// TwinCAT 3 PLC project Punzonatrice01
// ProgramVersion: 3.1.4024.0
// libraries:
//   Tc2_Standard, * (Beckhoff Automation GmbH)
//   Tc2_System, * (Beckhoff Automation GmbH)
//   Tc3_Module, * (Beckhoff Automation GmbH)
//   Util, * (System)
// project tree:
//   DUTs/ tStatiMSF.TcTLEO
//   GVLs/ GVL_IO.TcGVL
//   / PlcTask.TcTTO
//   POUs/ MAIN.TcPOU
//   POUs/MSF/FB/ FB_Blink.TcPOU, FB_MSF.TcPOU
// real-time tasks:
//   TASK PlcTask: cycle T#10ms, priority 20, ADS port 350
// motion (NC):
//   TASK NC-Task 1 SAF: cycle T#2ms, priority 4, ADS port 501
//   TASK NC-Task 1 SVB: cycle T#10ms, priority 8, ADS port 511
//   AXIS Asse 1 (id 1)
//     OtherSettings: AllowMotionCmdToSlave=true
//     encoder EncType=4
//       EncPara: MaxCount=#x0000ffff
//         Inc: RefSoftSyncMask=#x0000ffff
//     drive DrvType=24
//       Analog: TorqueSetpointScale=10, ScaleFactorActTorque=0.1
//       TimeComp: TaskDelayCycles=1
//     controller CtrType=1
//       CtrPara: PriorControlFactor=1
//         Observer: BandWidth=20
// I/O:
//   DEVICE Dispositivo 1 (EtherCAT), AmsNetId 192.168.17.154.2.1
//     Terminale 1 (EK1200) [EK1200-5000 EtherCAT Power supply (2A E-Bus)]
//       Terminale 2 (EL1809) [EL1809 16Ch. Dig. Input 24V, 3ms]
//       Terminale 3 (EL2809) [EL2809 16Ch. Dig. Output 24V, 0.5A]
//       Terminale 4 (EL3201) [EL3201 1Ch. Ana. Input PT100 (RTD)]
//       Terminale 5 (EL3311) [EL3311 1Ch. Ana. Input Thermocouple (TC)]
//       Terminale 6 (EL3004) [EL3004 4Ch. Ana. Input +/-10V]
//       Terminale 7 (EL1918) [EL1918, 8Ch. Safety Input 24V, TwinSAFE]
//         modules: Module 1 (FSOE), Module 2 (FSLOGIC)
//       Terminale 8 (EL2904) [EL2904, 4 Ch. Safety Output 24V, 0.5A, TwinSAFE]
//         modules: Module 1 (FSOES), Module 2 (DO)
//       Terminale 9 (EL9011) [EL9011 End Terminal]
//   DEVICE Dispositivo 4 (EtherCAT), AmsNetId 192.168.17.154.5.1
//     Terminale 10 (EK1100) [EK1100 EtherCAT Coupler (2A E-Bus)]
//       Terminale 11 (EL1809) [EL1809 16Ch. Dig. Input 24V, 3ms]
//       Terminale 12 (EL2809) [EL2809 16Ch. Dig. Output 24V, 0.5A]
//       Terminale 13 (EL1809) [EL1809 16Ch. Dig. Input 24V, 3ms]
//       Terminale 14 (EL2809-0015) [EL2809-0015 16Ch. Dig. Output 24V DC, 0.35A, not short-circuit proof]
//       Terminale 15 (EL7031) [EL7031 1Ch. Stepper motor output stage (24V, 1.5A)]
//       Terminale 7 (EL9011) [EL9011 End Terminal]
// variable links:
//   NC-Task 1 SAF/Axes/Asse 1 <-> Device 4 (EtherCAT)/Term 10 (EK1100)/Term 15 (EL7031)
//     Drive/Inputs/In/nState1 @bit 3 <-> STM Status/Status/Error
//     Drive/Inputs/In/nState1 @bit 5 <-> STM Status/Status/Moving negative
//     Drive/Inputs/In/nState1 @bit 4 <-> STM Status/Status/Moving positive
//     Drive/Inputs/In/nState1 @bit 1 <-> STM Status/Status/Ready
//     Drive/Inputs/In/nState1 <-> STM Status/Status/Ready to enable
//     Drive/Inputs/In/nState1 @bit 6 <-> STM Status/Status/Torque reduced
//     Drive/Inputs/In/nState1 @bit 2 <-> STM Status/Status/Warning
//     Drive/Inputs/In/nState2 @bit 3 <-> STM Status/Status/Digital input 1
//     Drive/Inputs/In/nState2 @bit 4 <-> STM Status/Status/Digital input 2
//     Drive/Inputs/In/nState2 @bit 5 <-> STM Status/Status/Sync error
//     Drive/Inputs/In/nState2 @bit 7 <-> STM Status/Status/TxPDO Toggle
//     Drive/Inputs/In/nState4 @bit 1 <-> WcState/InputToggle
//     Drive/Inputs/In/nState4 <-> WcState/WcState
//     Drive/Outputs/Out/nCtrl1 <-> STM Control/Control/Enable
//     Drive/Outputs/Out/nCtrl1 @bit 2 <-> STM Control/Control/Reduce torque
//     Drive/Outputs/Out/nCtrl1 @bit 1 <-> STM Control/Control/Reset
//     Drive/Outputs/Out/nDataOut2[0] <-> STM Velocity/Velocity
//     Enc/Inputs/In/nDataIn1[0] <-> ENC Status compact/Counter value
//     Enc/Inputs/In/nDataIn2[0] <-> ENC Status compact/Latch value
//     Enc/Inputs/In/nState1 @bit 4 <-> ENC Status compact/Status/Counter overflow
//     Enc/Inputs/In/nState1 @bit 3 <-> ENC Status compact/Status/Counter underflow
//     Enc/Inputs/In/nState1 @bit 1 <-> ENC Status compact/Status/Latch extern valid
//     Enc/Inputs/In/nState1 @bit 2 <-> ENC Status compact/Status/Set counter done
//     Enc/Inputs/In/nState2 @bit 4 <-> ENC Status compact/Status/Status of extern latch
//     Enc/Inputs/In/nState2 @bit 5 <-> ENC Status compact/Status/Sync error
//     Enc/Inputs/In/nState2 @bit 7 <-> ENC Status compact/Status/TxPDO Toggle
//     Enc/Inputs/In/nState4 @bit 1 <-> WcState/InputToggle
//     Enc/Inputs/In/nState4 <-> WcState/WcState
//     Enc/Outputs/Out/nCtrl1 @bit 3 <-> ENC Control compact/Control/Enable latch extern on negative edge
//     Enc/Outputs/Out/nCtrl1 @bit 1 <-> ENC Control compact/Control/Enable latch extern on positive edge
//     Enc/Outputs/Out/nCtrl1 @bit 2 <-> ENC Control compact/Control/Set counter
//     Enc/Outputs/Out/nDataOut1[0] <-> ENC Control compact/Set counter value
//   Punzonatrice01/Punzonatrice01 Instance <-> Device 1 (EtherCAT)/Term 1 (EK1200)/Term 2 (EL1809)
//     PlcTask Inputs/GVL_IO.Ack <-> Channel 7/Input
//     PlcTask Inputs/GVL_IO.Emg <-> Channel 8/Input
//     PlcTask Inputs/GVL_IO.I{1..4} <-> Channel {1..4}/Input  (4 links)
//     PlcTask Inputs/GVL_IO.Start <-> Channel 5/Input
//     PlcTask Inputs/GVL_IO.Stop <-> Channel 6/Input
//   Punzonatrice01/Punzonatrice01 Instance <-> Device 1 (EtherCAT)/Term 1 (EK1200)/Term 3 (EL2809)
//     PlcTask Outputs/GVL_IO.L_ACK <-> Channel 7/Output
//     PlcTask Outputs/GVL_IO.L_START <-> Channel 5/Output
//     PlcTask Outputs/GVL_IO.L_STOP <-> Channel 6/Output
//     PlcTask Outputs/GVL_IO.Q{1..4} <-> Channel {1..4}/Output  (4 links)

CONFIGURATION Punzonatrice01
    RESOURCE PLC ON TwinCAT3
        TASK PlcTask(INTERVAL := T#10ms, PRIORITY := 20);
        PROGRAM MAIN WITH PlcTask : MAIN;
    END_RESOURCE
END_CONFIGURATION

// ---- DUTs/tStatiMSF.TcTLEO
{attribute 'qualified_only'}
{attribute 'strict'}
TYPE tStatiMSF :
(
	S0_Spento := 0,
	S1_RipristinoMandrino,
	S2_AttesaPezzo,
	S3_PausaIngresso,
	S4_Caricamento,
	S5_DiscesaMandrino,
	S6_SalitaMandrino,
	S7_Scarico,
	S8_PausaScarico,
	SE_Emergenza,
	SA1_RipristinoMAndrino,
	SA2_UscitaPezzo
);
END_TYPE

// ---- GVLs/GVL_IO.TcGVL
{attribute 'qualified_only'}
VAR_GLOBAL
	// sensori bordo macchina
    I1    AT %I*    :    BOOL;
    I2    AT %I*    :    BOOL;
    I3    AT %I*    :    BOOL;
    I4    AT %I*    :    BOOL;
    // pulsanti di comando
    Start    AT %I*    :    BOOL;
    Stop    AT %I*    :    BOOL;
    Ack        AT %I*    :    BOOL;
    Emg        AT %I*    :    BOOL;
 
    // attuatori
    Q1    AT %Q*    :    BOOL;
    Q2    AT %Q*    :    BOOL;
    Q3    AT %Q*    :    BOOL;
    Q4    AT %Q*    :    BOOL;
    // indicatori pannello operatore
    L_START    AT %Q*    :    BOOL;
    L_STOP    AT %Q*    :    BOOL;
    L_ACK    AT %Q*    :    BOOL;    
END_VAR

// ---- POUs/MAIN.TcPOU
PROGRAM MAIN
VAR
	nastro1	: FB_MSF();
	
END_VAR

nastro1(
	I1:= GVL_IO.I1, 
	I2:= GVL_IO.I2, 
	I3:= GVL_IO.I3, 
	I4:= GVL_IO.I4, 
	Start:= GVL_IO.Start, 
	Stop:= GVL_IO.Stop, 
	Ack:= GVL_IO.Ack, 
	Emg:= GVL_IO.Emg, 
	Q1=> GVL_IO.Q1, 
	Q2=> GVL_IO.Q2, 
	Q3=> GVL_IO.Q3, 
	Q4=> GVL_IO.Q4, 
	L_START=> GVL_IO.L_START, 
	L_STOP=> GVL_IO.L_STOP, 
	L_ACK=> GVL_IO.L_ACK);

END_PROGRAM

// ---- POUs/MSF/FB/FB_MSF.TcPOU
FUNCTION_BLOCK FB_MSF
VAR_INPUT
	// sensori bordo macchina
	I1		:	BOOL;
	I2		: 	BOOL;
	I3		:	BOOL;
	I4		: 	BOOL;
	
	// pulsanti di comando
	Start	: 	BOOL;
	Stop	:	BOOL;
	Ack		: 	BOOL;
	Emg		: 	BOOL;
	
END_VAR
VAR_OUTPUT
	// attuatori
	Q1		:	BOOL;
	Q2		:	BOOL;
	Q3		:	BOOL;
	Q4		:	BOOL;

	// indicatori pannello indicatore
	L_START	: 	BOOL;
	L_STOP	: 	BOOL;
	L_ACK	: 	BOOL;
END_VAR
VAR
	// abilitazione := Stop AND Emg;
	enable 	:	BOOL;
	
	// variabile di stato
	stato	:	tStatiMSF	:=	tStatiMSF.S0_Spento;
	
	// timer per gli stati
	T34		: 	TON();
	T82		:	TON();
	TE		:	TON();
	TA		:	TON();
	
	// lampeggiatore
	osc		: 	FB_Blink();
	fbBlink :   BLINK;
	// richiesta di arresto a fine ciclo
	mArresto	:	BOOL;

	// pezzo carico
	mPezzoCarico	:	BOOL;
	// transizione S0->S1
	tr_S0_S1	: 	BOOL;
	// transizione S0->S1
	tr_S0_S2	: 	BOOL;
	// transizione S1->S0
	tr_S1_S0	:	BOOL;
	// transizione S1->S2
	tr_S1_S2	: 	BOOL;
	//transizione da S2->S3
	tr_S2_S0	:	BOOL;
	// transizione S2->S3
	tr_S2_S3	: 	BOOL;
	// transizione S3->S4
	tr_S3_S4	: 	BOOL;
	// transizione S4->S5
	tr_S4_S5	: 	BOOL;
	// transizione S4->S5
	tr_S4_SE	: 	BOOL;
	// transizione S5->S6
	tr_S5_S6	: 	BOOL;
	// transizione S6->S7
	tr_S6_S7	: 	BOOL;
	// transizione S7->S8
	tr_S7_S8	: 	BOOL;
	// transizione S7->SE
	tr_S7_SE	: 	BOOL;
	// transizione S8->S0
	tr_S8_S0	: 	BOOL;
	// transizione S8->S2
	tr_S8_S2	: 	BOOL;
	// transizione SE->SA
	tr_SE_SA1	: 	BOOL;
	// transizione SA1->SA2
	tr_SA1_SA2	: 	BOOL;
	// transizione SA2->S0
	tr_SA2_S0	: 	BOOL;
END_VAR

// 1. aggiornamento delle condizioni di abilitazione (stop, allatmi, ecc)
	enable	:=	Stop AND Emg;
	
// 2. aggiornamento di timers, contatori, triggers sui fronti
	T34( IN := (stato = tStatiMSF.S3_PausaIngresso), PT := T#2S );
	T82( IN := (stato = tStatiMSF.S8_PausaScarico), PT := T#3S );
	TE( IN := (stato = tStatiMSF.S4_Caricamento), PT := T#5S );
	TE( IN := (stato = tStatiMSF.S7_Scarico), PT := T#5S );
	TE( IN := (stato = tStatiMSF.SA2_UscitaPezzo), PT := T#5S );
	TA( IN := (stato = tStatiMSF.SA1_RipristinoMandrino), PT := T#2S );
	osc(enable := TRUE, t_high := T#1S, t_low := T#500MS);
// 3. valutazione della condizione di arresto nominale
	IF( Stop = FALSE AND Emg = TRUE ) THEN 
		mArresto := TRUE;
	END_IF
	
// 4. valutazione della condizione di arresto di emergenza
	IF( Emg = FALSE AND (stato <> tStatiMSF.S0_Spento)) THEN
		stato := tStatiMSF.SE_Emergenza;
	END_IF
	
	
// 5. aggiornamento delle condizioni di transito di stato
	tr_S0_S1 :=	NOT(I3) AND Start AND enable;
	// transizione S0->S2
	tr_S0_S2 := I3 AND Start AND enable; 
	// transizione S1->S0
	tr_S1_S0 := mArresto AND Emg;	
	// transizione S1->S2
	tr_S1_S2 := I3 AND Emg;
	//transizione da S2->S3
	tr_S2_S0 := mArresto AND Emg;
	// transizione S2->S3
	tr_S2_S3 := NOT(I1) AND Emg;
	// transizione S3->S4
	tr_S3_S4 := T34.Q AND NOT(I1) AND Emg;
	// transizione S4->S5
	tr_S4_S5 := NOT(I2) AND Emg; 
	// transizione S4->S5
	tr_S4_SE := TE.Q AND Emg;	
	// transizione S5->S6
	tr_S5_S6 := I4 AND Emg; 
	// transizione S6->S7
	tr_S6_S7 := I3 AND Emg;
	// transizione S4->S5
	tr_S7_SE := TE.Q AND Emg;
	// transizione S7->S8
	tr_S7_S8 := NOT(I1) AND Emg;
	// transizione S8->S0
	tr_S8_S0 := mArresto AND Emg ;
	// transizione S8->S2
	tr_S8_S2 := T82.Q AND NOT(mArresto) AND I1 AND enable;
	// transizione SE->SA
	tr_SE_SA1 := EMG AND Ack;
	// transizione SE->SA
	tr_SA1_SA2 := TA.Q;
	// transizione SA->S0
	tr_SA2_S0 := (mPezzoCarico AND NOT(I1) AND I3) OR (NOT(mPezzoCarico) AND I3)OR(TE.Q);

// 6. switch-case della MSF
	CASE stato OF
	tStatiMSF.S0_Spento:
	

    // comando uscite
	L_START := FALSE;
	L_STOP := TRUE;
	L_ACK := FALSE;
	Q1 := FALSE;
	Q2 := FALSE;
	Q3 := FALSE;
	Q4 := FALSE;
	// reset memoria
	mArresto := FALSE;
	mPezzoCarico := FALSE;
	IF tr_S0_S1 THEN
		stato := tStatiMSF.S1_RipristinoMandrino;
	ELSIF tr_S0_S2 THEN
		stato := tStatiMSF.S2_AttesaPezzo;
	END_IF
	
	tStatiMSF.S1_RipristinoMandrino:
	// comando uscite
	L_START := TRUE;
	L_STOP := FALSE;
	L_ACK := osc.q;// lamepggio
	Q1 := FALSE;
	Q2 := FALSE;
	Q3 := NOT(I3);
	Q4 := FALSE;
	// set memoria
	mPezzoCarico := FALSE;
	IF tr_S1_S2 THEN
		stato := tStatiMSF.S2_AttesaPezzo;
	ELSIF tr_S1_S0 THEN
		stato := tStatiMSF.S0_Spento;
	END_IF
	
	tStatiMSF.S2_AttesaPezzo:
	// comando uscite
	L_START := TRUE;
	L_STOP := FALSE;
	L_ACK := FALSE;
	Q1 := FALSE;
	Q2 := FALSE;
	Q3 := FALSE;
	Q4 := FALSE;
	// set memoria
	mPezzoCarico := FALSE;
	IF tr_S2_S3 THEN
		stato := tStatiMSF.S3_PausaIngresso;
	ELSIF tr_S2_S0 THEN
		stato := tStatiMSF.S0_Spento;
	END_IF
	
	tStatiMSF.S3_PausaIngresso:
	// comando uscite
	L_START := TRUE;
	L_STOP := FALSE;
	L_ACK := FALSE;
	Q1 := FALSE;
	Q2 := FALSE;
	Q3 := FALSE;
	Q4 := FALSE;
	// set memoria
	mPezzoCarico := TRUE;
	IF tr_S3_S4 THEN
		stato := tStatiMSF.S4_Caricamento;
	END_IF
	
	tStatiMSF.S4_Caricamento:
	// comando uscite
	L_START := TRUE;
	L_STOP := FALSE;
	L_ACK := FALSE;
	Q1 := TRUE;
	Q2 := FALSE;
	Q3 := FALSE;
	Q4 := FALSE;
	// set memoria
	mPezzoCarico := TRUE;
	IF tr_S4_S5 THEN
		stato := tStatiMSF.S5_DiscesaMandrino;
	ELSIF tr_S4_SE THEN
		stato := tStatiMSF.SE_Emergenza;
	 
	END_IF
	
	tStatiMSF.S5_DiscesaMandrino:
	// comando uscite
	L_START := TRUE;
	L_STOP := FALSE;
	L_ACK := FALSE;
	Q1 := FALSE;
	Q2 := FALSE;
	Q3 := FALSE;
	Q4 := NOT(I4);
	// set memoria
	mPezzoCarico := TRUE;
	IF tr_S5_S6 THEN
		stato := tStatiMSF.S6_SalitaMandrino;
	END_IF
		
	tStatiMSF.S6_SalitaMandrino:
	// comando uscite
	L_START := TRUE;
	L_STOP := FALSE;
	L_ACK := FALSE;
	Q1 := FALSE;
	Q2 := FALSE;
	Q3 := NOT(I3);
	Q4 := FALSE;
	// set memoria
	mPezzoCarico := TRUE;
	IF tr_S6_S7 THEN
		stato := tStatiMSF.S7_Scarico;
	END_IF
		
	tStatiMSF.S7_Scarico:
	// comando uscite
	L_START := TRUE;
	L_STOP := FALSE;
	L_ACK := FALSE;
	Q1 := FALSE;
	Q2 := TRUE;
	Q3 := FALSE;
	Q4 := FALSE;
	// set memoria
	mPezzoCarico := TRUE;
	IF tr_S7_S8 THEN
		stato := tStatiMSF.S8_PausaScarico;
	ELSIF tr_S7_SE THEN
		stato := tStatiMSF.SE_Emergenza;
	END_IF
		
	tStatiMSF.S8_PausaScarico:
	// comando uscite
	L_START := TRUE;
	L_STOP := FALSE;
	L_ACK := FALSE;
	Q1 := FALSE;
	Q2 := FALSE;
	Q3 := FALSE;
	Q4 := FALSE;
	// set memoria
	mPezzoCarico := FALSE;
	IF tr_S8_S0 THEN
		stato := tStatiMSF.S0_Spento;
	ELSIF tr_S8_S2 THEN
		stato := tStatiMSF.S2_AttesaPezzo;
	END_IF
		
	tStatiMSF.SE_Emergenza:
	// comando uscite
	L_START := TRUE;
	L_STOP := osc.q; // lampeggio
	L_ACK := TRUE;
	Q1 := FALSE;
	Q2 := FALSE;
	Q3 := FALSE;
	Q4 := FALSE;

	IF tr_SE_SA1 THEN
		stato := tStatiMSF.SA1_RipristinoMandrino;
	END_IF
		
	tStatiMSF.SA1_RipristinoMandrino:
	// comando uscite
	L_START := TRUE;
	L_STOP := FALSE;
	L_ACK := osc.q; // lampeggio
	Q1 := FALSE;
	Q2 := FALSE;
	Q3 := NOT(I3);
	Q4 := FALSE;
	
	IF tr_SA1_SA2 THEN
		stato := tStatiMSF.SA2_UscitaPezzo;
	END_IF

	tStatiMSF.SA2_UscitaPezzo:
	// comando uscite
	L_START := TRUE;
	L_STOP := FALSE;
	L_ACK := osc.q; // lampeggio
	Q1 := FALSE;
	Q2 := mPezzoCarico;
	Q3 := FALSE;
	Q4 := FALSE;
	
	IF tr_SA2_S0 THEN
		stato := tStatiMSF.S0_Spento;
	END_IF
ELSE
	stato := tStatiMSF.SE_Emergenza;
END_CASE

END_FUNCTION_BLOCK

// ---- POUs/MSF/FB/FB_Blink.TcPOU
FUNCTION_BLOCK FB_Blink
VAR_INPUT
	enable	:	BOOL;
	t_high	:	TIME;
	t_low	:	TIME;
	
END_VAR
VAR_OUTPUT
	q	:	BOOL;
END_VAR
VAR
	T1		: 	TON();
	T2		:	TON();
END_VAR

T1(IN := (enable AND NOT(T2.Q ) ), PT := t_low);
T2(IN := T1.Q, PT	:= t_high ); 
q := T1.Q;

END_FUNCTION_BLOCK
